// LS Electric XG5000 project: 유튜브방송용_2021082321
// PLC NewPLC

PROGRAM NewProgram (task: 스캔 프로그램)

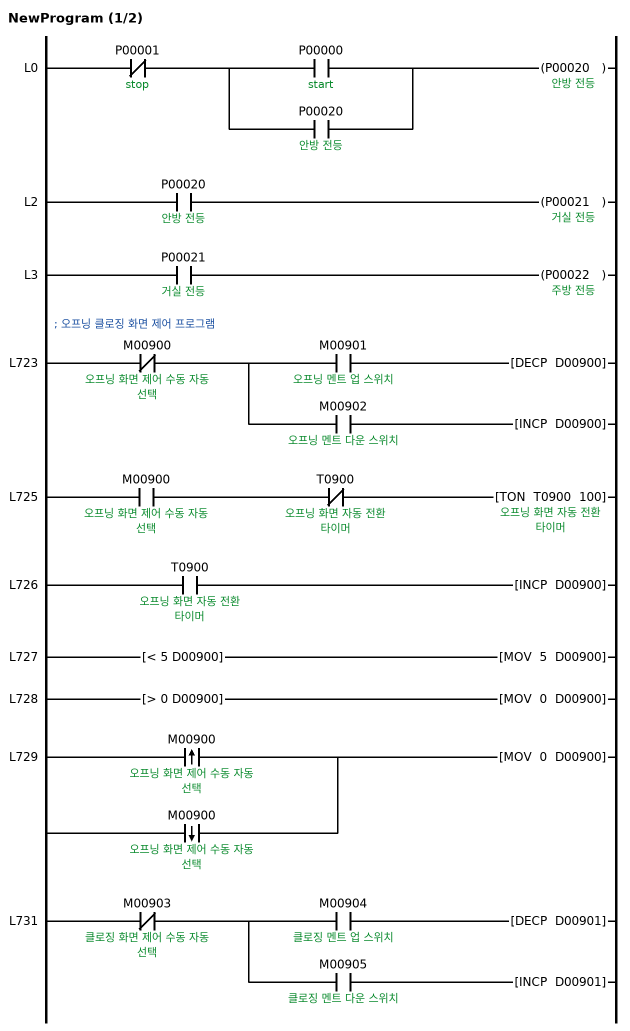
; L0
LOAD NOT  P00001	// stop
LOAD      P00000	// start
OR        P00020	// 안방 전등
AND LOAD
OUT       P00020	// 안방 전등
; L2
LOAD      P00020	// 안방 전등
OUT       P00021	// 거실 전등
; L3
LOAD      P00021	// 거실 전등
OUT       P00022	// 주방 전등
// 오프닝 클로징 화면 제어 프로그램
; L723
LOAD NOT  M00900	// 오프닝 화면 제어 수동 자동 선택
MPUSH
AND       M00901	// 오프닝 멘트 업 스위치
DECP      D00900
MPOP
AND       M00902	// 오프닝 멘트 다운 스위치
INCP      D00900
; L725
LOAD      M00900	// 오프닝 화면 제어 수동 자동 선택
AND NOT   T0900	// 오프닝 화면 자동 전환 타이머
TON       T0900 100	// 오프닝 화면 자동 전환 타이머
; L726
LOAD      T0900	// 오프닝 화면 자동 전환 타이머
INCP      D00900
; L727
LOAD<     5 D00900
MOV       5 D00900
; L728
LOAD>     0 D00900
MOV       0 D00900
; L729
LOADP     M00900	// 오프닝 화면 제어 수동 자동 선택
ORN       M00900	// 오프닝 화면 제어 수동 자동 선택
MOV       0 D00900
; L731
LOAD NOT  M00903	// 클로징 화면 제어 수동 자동 선택
MPUSH
AND       M00904	// 클로징 멘트 업 스위치
DECP      D00901
MPOP
AND       M00905	// 클로징 멘트 다운 스위치
INCP      D00901

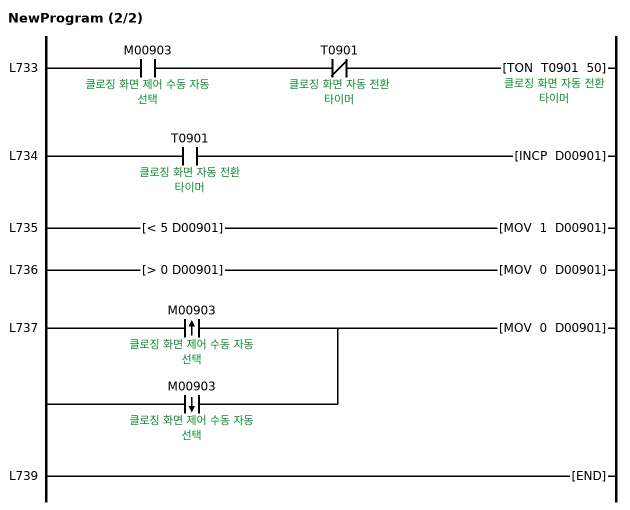
; L733
LOAD      M00903	// 클로징 화면 제어 수동 자동 선택
AND NOT   T0901	// 클로징 화면 자동 전환 타이머
TON       T0901 50	// 클로징 화면 자동 전환 타이머
; L734
LOAD      T0901	// 클로징 화면 자동 전환 타이머
INCP      D00901
; L735
LOAD<     5 D00901
MOV       1 D00901
; L736
LOAD>     0 D00901
MOV       0 D00901
; L737
LOADP     M00903	// 클로징 화면 제어 수동 자동 선택
ORN       M00903	// 클로징 화면 제어 수동 자동 선택
MOV       0 D00901
; L739
END

VARIABLES AND COMMENTS (devices not used above)
P00002	BIT	주방 스위치